RESOURCE_TYPE EMB_RES (* Most basic resource for executing FB networks *)
  (* Function: This resource provides the most basic functionality of an IEC 61499 resource, namely executing FB networks. For convenience it already contains an instance of the E_RESTART FB providing events for starting up and shutting down an application. This resource is based on examples found in the different parts of IEC 61499 and the documentation at http://www.holobloc.com/doc/fb/rt/EMB_RES.htm; Description: Copyright (c) 2017 fortiss GmbH This program and the accompanying materials are made available under the terms of the Eclipse Public License 2.0 which is available at https://www.eclipse.org/legal/epl-2.0/ SPDX-License-Identifier: EPL-2.0 *)
  (* Version 1.0, 2017-12-02, Alois Zoitl, fortiss GmbH *)
  (* Version 3.0, 2025-04-14, Patrick Aigner, changed package *)
  PACKAGE iec61499::system;
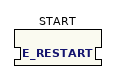
  FBS
    START : iec61499::events::E_RESTART;
  END_FBS
END_RESOURCE_TYPE
